FUNCTION_BLOCK SpacerRecollectionUnit //EXTENDS SectionEx
VAR_IN_OUT
	robot : RobotA26; //placeholder, will need another robot definition for A26
	robotSlider : ServoNC;
END_VAR
VAR_INPUT
	spacerPresent_A24_LRC_C02 : BOOL; //these conveyoors move bundles from A2.7 to A2.4
	spacerPresent_A24_LRC_C04 : BOOL;
	spacerPresent_A24_LRC_C06 : BOOL;
	spacerPresent_A24_LRC_C08 : BOOL;
	spacerPresent_A24_LRC_C10 : BOOL;
	spacerPresent_A24_LRC_C12 : BOOL;
END_VAR
VAR_OUTPUT
	ready : BOOL;
	busy : BOOL;
	done : BOOL;
	error : BOOL;
	
	failCounter : INT;
END_VAR
VAR
	//spacersPresent : ARRAY[1..6] OF BOOL;
	
	step : (IDLE, PICK_SPACER, COMPLETE);
	iPosition : INT;
END_VAR

ready := step = 0;
busy := step > 0;
done := done;
error := error;
(*
spacersPresent[1] := spacerPresent_A24_LRC_C02;
spacersPresent[2] := spacerPresent_A24_LRC_C04;
spacersPresent[3] := spacerPresent_A24_LRC_C06;
spacersPresent[4] := spacerPresent_A24_LRC_C08;
spacersPresent[5] := spacerPresent_A24_LRC_C10;
spacersPresent[6] := spacerPresent_A24_LRC_C12;
*)
IF 
	A24.A24_SC_C01.IsOccupied OR
	A24.A24_SC_C03.IsOccupied OR
	A24.A24_SC_C05.IsOccupied OR
	A24.A24_SC_C07.IsOccupied OR
	A24.A24_SC_C09.IsOccupied OR
	A24.A24_SC_C11.IsOccupied OR
	A24.A24_SC_C13.IsOccupied
THEN
	robot.clearCommand();
	
ELSE
	//remove spacers from transfer conveyors in ascending order
	process();
	
END_IF

METHOD process : BOOL
VAR_INPUT
END_VAR
VAR
	spacersPresent : ARRAY[1..6] OF BOOL := [
		spacerPresent_A24_LRC_C02,
		spacerPresent_A24_LRC_C04,
		spacerPresent_A24_LRC_C06,
		spacerPresent_A24_LRC_C08,
		spacerPresent_A24_LRC_C10,
		spacerPresent_A24_LRC_C12];
END_VAR
VAR CONSTANT
	suctionDistance : INT := 10;
END_VAR
{warning disable C0371}

iPosition := MAX(1, iPosition); //value is always at least 1

CASE step OF
	IDLE:
		IF DataIsEmpty(arr := ADR(spacersPresent), arrSize := SIZEOF(spacersPresent)) THEN
			iPosition := 0;
			failCounter := 0;
			process := TRUE;
		
		ELSIF NOT spacersPresent[iPosition] THEN
			iPosition := iPosition + 1;
			
		ELSIF robot.Ready THEN
			step := PICK_SPACER;
		END_IF
		
	PICK_SPACER:
		IF robot.eoatDistance > suctionDistance THEN
			robot.HoldMaterial := 'SPACER';
		ELSE
			robot.HoldMaterial := '';
		END_IF
	
		IF robot.Done THEN
			step := COMPLETE;
		ELSE
			robot.setGroup(group := 1, value := TaskA26.PICK_SPACER);
			robot.setGroup(group := 2, value := iPosition);
		END_IF
		
	COMPLETE:
		robot.HoldMaterial := '';
		
		IF spacersPresent[iPosition] THEN
			failCounter := failCounter + 1;
		END_IF
		
		robot.clearCommand();
		step := 0;
	
END_CASE
END_METHOD

END_FUNCTION_BLOCK

(* stored: Version 1.1.0.1, ProductVersion 3.1.4024.11
   POU SpacerRecollectionUnit: Id {6fea2dc6-ce06-4fa1-9588-ba3bbddda180}, SpecialFunc None
   Method process: Id {0707ef1b-9ba5-4d26-b34d-69bdd29b3450} *)
